SUBAPPLICATION Uebung_073 (* VDS auf UT ausgeben *)
  (* Standard: 61499-2 *)
  (* Version 1.0, 2023-10-23, franz *)
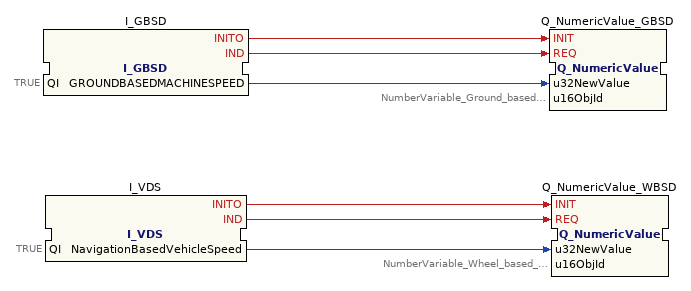
  FBS
    I_GBSD : I_GBSD(QI := TRUE);
    Q_NumericValue_GBSD : Q_NumericValue(u16ObjId := NumberVariable_Ground_based_machine_speed);
    I_VDS : I_VDS(QI := TRUE);
    Q_NumericValue_WBSD : Q_NumericValue(u16ObjId := NumberVariable_Wheel_based_machine_speed);
  END_FBS
  EVENT_CONNECTIONS
    I_GBSD.INITO TO Q_NumericValue_GBSD.INIT;
    I_GBSD.IND TO Q_NumericValue_GBSD.REQ;
    I_VDS.INITO TO Q_NumericValue_WBSD.INIT;
    I_VDS.IND TO Q_NumericValue_WBSD.REQ;
  END_CONNECTIONS
  DATA_CONNECTIONS
    I_GBSD.GROUNDBASEDMACHINESPEED TO Q_NumericValue_GBSD.u32NewValue;
    I_VDS.NavigationBasedVehicleSpeed TO Q_NumericValue_WBSD.u32NewValue;
  END_CONNECTIONS
END_SUBAPPLICATION
